// TIA Portal V19 export
TYPE "LTBSE_typeStatemachine"
TITLE = Typ Statemachinedata / Data for Statemachine
// Daten für Schrittkettenwerwaltung / Data
   STRUCT
      init : Bool;   // Init SQ / init sequence
      tap : Bool;   // Schrittkette Einzelschritt / tap next step
      auto : Bool;   // Automatik / Auto mode
      manual : Bool;   // Handbetrieb / manual mode
      state : DInt;   // aktueller Schritt
      stateNext : DInt;   // nächster Schritt / next step
      stateOld : DInt;   // vorhergehender Schritt / previos step
      s1 : Bool;   // Flanke kommender Schritt / rising Edge new state
      stepDiagText : WString[50];
      stepWaittime_1 : Struct   // Schrittwartezeit / waittime
         "timer" : IEC_TIMER;   // Timer / timer
         active : Bool;   // Zeit aktivieren / waittime active
         targettime : Real;   // [s] Zielzeit / [s] targettime
         expired : Bool;   // Zeit abgelaufen / waittime expired
      END_STRUCT;
      stepErrortime_1 : Struct   // Schrittfehlerzeit / error steptime
         "timer" : IEC_TIMER;   // Timer / timer
         active : Bool;   // Zeit aktivieren / errortime active
         targettime : Real;   // [s] Zielzeit / [s] targettime
         expired : Bool;   // Zeit abgelaufen / errortime expired
      END_STRUCT;
   END_STRUCT;
END_TYPE
